// TwinCAT 3 PLC project tc_mot_example
// ProgramVersion: 3.1.4022.7
// libraries:
//   lcls-twincat-motion, * (SLAC)
//   lcls2-cc-lib, * (SLAC)
//   PMPS, * (SLAC - LCLS)
//   Tc2_Standard, * (Beckhoff Automation GmbH)
//   Tc2_System, * (Beckhoff Automation GmbH)
//   Tc3_Module, * (Beckhoff Automation GmbH)
// project tree:
//   DUTs/ ENUM_Mirror_States.TcDUT
//   / PlcTask.TcTTO (not stored)
//   POUs/ Main.TcPOU
//   POUs/NewFolder1/ FB_Mirror_States.TcPOU
// real-time tasks:
//   TASK PlcTask: cycle T#10ms, priority 20, ADS port 350
// motion (NC):
//   TASK NC-Task 1 SAF: cycle T#2ms, priority 4, ADS port 501
//   TASK NC-Task 1 SVB: cycle T#10ms, priority 8, ADS port 511
//   AXIS M9X9 (id 1)
//   AXIS Example 2 Simulated Broken (id 2)
//   AXIS Example 3 Simulated Limits (id 3)
//   AXIS Example 4 PMPS (id 4)
// variable links:
//   tc_mot_example Instance <-> NC-Task 1 SAF/Axes/Example 2 Simulated Broken
//     PlcTask Inputs/Main.M2.Axis.NcToPlc <-> Outputs/ToPlc
//     PlcTask Outputs/Main.M2.Axis.PlcToNc <-> Inputs/FromPlc
//   tc_mot_example Instance <-> NC-Task 1 SAF/Axes/Example 3 Simulated Limits
//     PlcTask Inputs/Main.M3.Axis.NcToPlc <-> Outputs/ToPlc
//     PlcTask Outputs/Main.M3.Axis.PlcToNc <-> Inputs/FromPlc
//   tc_mot_example Instance <-> NC-Task 1 SAF/Axes/Example 4 PMPS
//     PlcTask Inputs/Main.M4.Axis.NcToPlc <-> Outputs/ToPlc
//     PlcTask Outputs/Main.M4.Axis.PlcToNc <-> Inputs/FromPlc
//   tc_mot_example Instance <-> NC-Task 1 SAF/Axes/M9X9
//     PlcTask Inputs/Main.M1.Axis.NcToPlc <-> Outputs/ToPlc
//     PlcTask Outputs/Main.M1.Axis.PlcToNc <-> Inputs/FromPlc

// ---- DUTs/ENUM_Mirror_States.TcDUT
TYPE ENUM_Mirror_States :
(
    Unknown := 0,
    In := 1,
    Out := 2
);
END_TYPE

// ---- POUs/Main.TcPOU
PROGRAM Main
VAR
    // Simulated motor that is always allowed to move
    {attribute 'pytmc' := '
        pv: M9X9:TST:MMS:XUP
        field: DESC Simulated Working Motor
    '}
    M1: DUT_MotionStage;
    fbMotion1: FB_MotionStageSim;
    
    {attribute 'pytmc' := '
      pv: M9X9:TST:MIRROR:STATE:SET
      io: i
    '}
    M9X9_Mirror_enumSet : ENUM_Mirror_States;
    {attribute 'pytmc' := '
     pv: M9X9:TST:MIRROR:STATE;
     io: i;
     field ZRST Unknown ;
     field ONST IN;
     field TWST OUT;
     '}
    
    fbM9X9_States: FB_Mirror_States := (
        bEnable := TRUE,
        sINtype := 'IN',
        nINPosition := 1100,
        fINDelta := 50,
        fINVelocity := 100
        );

    // Simulated motor that is never allowed to move
    {attribute 'pytmc' := '
        pv: PLC:TST:MOT:SIM:02
        field: DESC Simulated Broken Motor
    '}
    M2: DUT_MotionStage;
    fbMotion2: FB_MotionStage;

    // Simulated motor with limits at 0 and 100
    {attribute 'pytmc' := '
        pv: PLC:TST:MOT:SIM:03
        field: DESC Simulated Working Motor With Limits
    '}
    M3: DUT_MotionStage;
    fbMotion3: FB_MotionStage;
    
    // Simulated PPM motor with PMPS
    {attribute 'pytmc' := '
        pv: PLC:TST:MOT:SIM:04
        field: DESC Simulated PPM Motor
    '}
    M4: DUT_MotionStage;
    {attribute 'pytmc' := '
        pv: PLC:TST:MOT:SIM:04
    '}
    fbPPM: FB_PPM;
    
    // PMPS Machinery
    fbArbiterIO: FB_SubSysToArbiter_IO;
    {attribute 'pytmc' := 'pv: PLC:TST:MOT:ARB'}
    fbArbiter: FB_Arbiter(1);
    {attribute 'pytmc' := 'pv: PLC:TST:MOT:FFO:01'}
    fbFFHWO: FB_HardwareFFOutput := (bAutoReset := TRUE);
END_VAR

fbMotion1(stMotionStage := M1);
fbMotion2(stMotionStage := M2);

M3.bHardwareEnable := TRUE;
M3.bPowerSelf := TRUE;
M3.bLimitForwardEnable := M3.Axis.NcToPlc.ActPos < 99.7;
M3.bLimitBackwardEnable := M3.Axis.NcToPlc.ActPos > 0.2;

fbMotion3(stMotionStage := M3);

fbM9X9_States(
    enumSet := M9X9_Mirror_enumSet,
    stMotionStage := M1,
    fbArbiter := fbArbiter,
    fbFFHWO := fbFFHWO);
    
M9X9_Mirror_enumSet := fbM9X9_States.setState;

M4.bHardwareEnable := TRUE;
M4.bPowerSelf := FALSE;
M4.bLimitForwardEnable := TRUE;
M4.bLimitBackwardEnable := TRUE;

fbPPM.nTransitionAssertionID := 16#2FF0;
fbPPM.nUnknownAssertionID := 16#2FF9;
fbPPM.stOut.fPosition := -10;
fbPPM.stOut.bUseRawCounts := FALSE;
fbPPM.stOut.nRequestAssertionID := 16#2FF1;
fbPPM.stOut.stBeamParams := PMPS_GVL.cstFullBeam;
fbPPM.stOut.bValid := TRUE;
fbPPM.stPower.fPosition := -50;
fbPPM.stPower.bUseRawCounts := FALSE;
fbPPM.stPower.nRequestAssertionID := 16#2FF2;
fbPPM.stPower.stBeamParams := PMPS_GVL.cstFullBeam;
fbPPM.stPower.bValid := TRUE;
fbPPM.stYag1.fPosition := -70;
fbPPM.stYag1.bUseRawCounts := FALSE;
fbPPM.stYag1.nRequestAssertionID := 16#2FF3;
fbPPM.stYag1.stBeamParams := PMPS_GVL.cstFullBeam;
fbPPM.stYag1.bValid := TRUE;
fbPPM.stYag2.fPosition := -100;
fbPPM.stYag2.bUseRawCounts := FALSE;
fbPPM.stYag2.nRequestAssertionID := 16#2FF4;
fbPPM.stYag2.stBeamParams := PMPS_GVL.cstFullBeam;
fbPPM.stYag2.bValid := TRUE;

fbPPM(
    stYStage:=M4,
    fbArbiter:=fbArbiter,
    fbFFHWO:=fbFFHWO,
    );
    
fbFFHWO.Execute();
fbArbiterIO(
    Arbiter:=fbArbiter,
    fbFFHWO:=fbFFHWO);

END_PROGRAM

// ---- POUs/NewFolder1/FB_Mirror_States.TcPOU
FUNCTION_BLOCK FB_Mirror_States EXTENDS FB_PositionStateBase_WithPMPS
VAR_INPUT
    enumSet : INT;
    stM9X9 : DUT_PositionState;
    sINtype : STRING := '';
    nINPosition : UDINT;
    fINDelta : LREAL;
    fINVelocity : LREAL;
    
    
END_VAR
VAR_OUTPUT
    {attribute 'pytmc' := '
      pv : GET
      io : i
    '}
    enumGet : ENUM_Mirror_States;
  END_VAR
VAR
    bInitState : BOOL := TRUE;
END_VAR

if bInitState THEN
    bInitState := FALSE;
    stM9X9.bUseRawCounts := FALSE;
    stM9X9.bMoveOk := TRUE;
    stM9X9.bValid := TRUE;
    //stM9X9.nRequestAssertionID := nTransitionAssertionID + 1;
    stM9X9.sName := sINtype;
    stM9X9.fPosition := nINPosition;
    stM9X9.fDelta := fINDelta;
    stM9X9.fVelocity := fINVelocity;
    
    arrStates[1] := stM9X9;
END_IF

setState := enumSet;
Exec();
enumGet := getState;
enumSet := setState;

END_FUNCTION_BLOCK
